FUNCTION_BLOCK FB_TOR_ES EXTENDS FB_TOR_Base
//////////////////
//  Emergency stop system
//////////////////
VAR_INPUT PERSISTENT
	// Parameters of the Object (instance/model specific) 
	ParamTempoEs :TIME:=T#2S;	// (s) Tempo before raising an alarm
END_VAR

VAR_OUTPUT
	//Child objects
	
END_VAR

VAR_INPUT
	// I/O Inputs 		                                     				
		
	
END_VAR

VAR
	//M_ALARMMANAGEMENT VARIABLES//
		FB_PermAlarm				: SR ;					// (NA) FB to maintain emergency stop Alarm 
		TON_ES						: TON ; 
 
	//M_STATEMANAGER VARIABLES//
		MesDataExd			: TOR_Standard ;  	
	// EMULATOR //
		Emul_MesState1				: BOOL;
		Emul_MesState2				: BOOL;
		
END_VAR

METHOD M_Execute
//////////////////
//  Method Calls 
/////////////////

VAR 
	// Method local variables (reinitialized at each cycle) 

END_VAR

	
	IF ParamNbSensors = 9 THEN // Use of contactor bi-stable No and NC
		IN_MesState2_IO := NOT IN_MesState2_IO;
	END_IF
SUPER^.M_Execute() ;
END_METHOD

END_FUNCTION_BLOCK

(* stored: Version 1.1.0.1, ProductVersion 3.1.4024.6
   POU FB_TOR_ES: Id {e731a6fc-fa21-4e89-878f-a8c68f7f3594}, SpecialFunc None
   Method M_Execute: Id {f380f390-cb8d-4c63-b849-bd3c65dc1d70} *)
